ABB RobotStudio station: Modulo_1.rspag

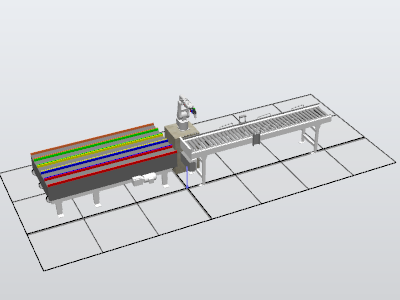
--- station ---
Station Prototipo1 (saved by RobotStudio 25.1.11133.0)
Controller Controlador1, task T_ROB1: task frame (RAPID world) sits at (289.3, 766.92, 800) mm, rotated rx 0 ry 0 rz -90 deg in the station
Controller Controlador1
  mechanical unit ROB_1: Robot1, 6 joints, base frame (0, 0, 0) mm
Layout (positions relative to the parent item):
  - Cinta entrada [part, from %ABB.RobotStudio.Models.Conveyors%\Conveyor Guide 400.rslib] at (77.15, 0, 0) mm
  - Apoyo1 [part], size 500 x 500 x 800 mm
  - Robot1 [mechanism, from %ABB.RobotStudio.Models.IRB120%\IRB120_3_58_G_01.rslib] at (289.3, 766.92, 800) mm, rotated rx 0 ry 0 rz -90 deg; joint values [0, 0, 0, 0, 0.5236, 0] (rad or m)
  - Apoyo cinta salida [part, from %ABB.RobotStudio.Models.Conveyors%\Conveyor 2400 3str h2.rslib] at (-191.15, 1159.17, 0) mm, rotated rx 0 ry 0 rz 180 deg
  - Estropajo_base [part] at (2748.27, 147.09, 782.53) mm, size 80 x 120 x 43 mm
  - Source [smart component, from Components\Source.rslib]
      properties: Source=Estropajo_base; Copy=(none); Parent=(none); Position=[2.748273 0.147093 0.782531]; Orientation=[0 0 0]; Transient=true; PhysicsBehavior=-1
  - LinearMover2 [smart component, from Components\LinearMover2.rslib]
      properties: Object=(none); Direction=[-1 0 0]; Distance=2.5; Duration=3; Reference=Global; ReferenceObject=(none)
  - Sink [smart component, from Components\Sink.rslib]
      properties: Object=(none)
  - Source_2 [smart component, from Components\Source.rslib]
      properties: Source=Estropajo_azul; Copy=(none); Parent=(none); Position=[2.748273 0.147093 0.782531]; Orientation=[0 0 0]; Transient=true; PhysicsBehavior=-1
  - Estropajo_azul [part] at (2748.27, 147.09, 782.53) mm, size 80 x 120 x 43 mm
  - Source_3 [smart component, from Components\Source.rslib]
      properties: Source=Estropajo_naranja; Copy=(none); Parent=(none); Position=[2.748273 0.147093 0.782531]; Orientation=[0 0 0]; Transient=true; PhysicsBehavior=-1
  - Source_4 [smart component, from Components\Source.rslib]
      properties: Source=Estropajo_amarillo; Copy=(none); Parent=(none); Position=[2.748273 0.147093 0.782531]; Orientation=[0 0 0]; Transient=true; PhysicsBehavior=-1
  - Source_6 [smart component, from Components\Source.rslib]
      properties: Source=Estropajo_verde; Copy=(none); Parent=(none); Position=[2.748273 0.147093 0.782531]; Orientation=[0 0 0]; Transient=true; PhysicsBehavior=-1
  - Estropajo_amarillo [part] at (2748.27, 147.09, 782.53) mm, size 80 x 120 x 43 mm
  - Estropajo_naranja [part] at (2748.27, 147.09, 782.53) mm, size 80 x 120 x 43 mm
  - Estropajo_verde [part] at (2748.27, 147.09, 782.53) mm, size 80 x 120 x 43 mm
  - Estropajo_5 [part] at (248.27, 147.09, 782.53) mm, size 80 x 120 x 43 mm
  - Estropajo_6 [part] at (-216.02, 245.91, 691.61) mm, size 80 x 120 x 43 mm
  - MyTool [mechanism, from Training Objects\myTool.rslib] at (289.3, 402.56, 1394) mm, rotated rx 180 ry 60 rz 90 deg
  - Attacher [smart component, from Components\Attacher.rslib]
      properties: Parent=MyTool; Flange=0; Child=(none); Mount=false; Offset=[0 0 0]; Orientation=[0 0 0]
  - Detacher [smart component, from Components\Detacher.rslib]
      properties: Child=(none); KeepPosition=true
  - Attacher_2 [smart component, from Components\Attacher.rslib]
      properties: Parent=MyTool; Flange=0; Child=(none); Mount=false; Offset=[0 0 0]; Orientation=[0 0 0]
  - Attacher_3 [smart component, from Components\Attacher.rslib]
      properties: Parent=MyTool; Flange=0; Child=(none); Mount=false; Offset=[0 0 0]; Orientation=[0 0 0]
  - Attacher_4 [smart component, from Components\Attacher.rslib]
      properties: Parent=MyTool; Flange=0; Child=(none); Mount=false; Offset=[0 0 0]; Orientation=[0 0 0]
  - Attacher_5 [smart component, from Components\Attacher.rslib]
      properties: Parent=MyTool; Flange=0; Child=(none); Mount=false; Offset=[0 0 0]; Orientation=[0 0 0]
  - LinearMover2_2 [smart component, from Components\LinearMover2.rslib]
      properties: Object=(none); Direction=[-1 0 0]; Distance=2.2; Duration=3; Reference=Global; ReferenceObject=(none)
  - Cinta entrada [part, from Components\Cinta salida.rslib] at (100, -50, 0) mm
Attachment: MyTool is attached to Robot1 / Link6
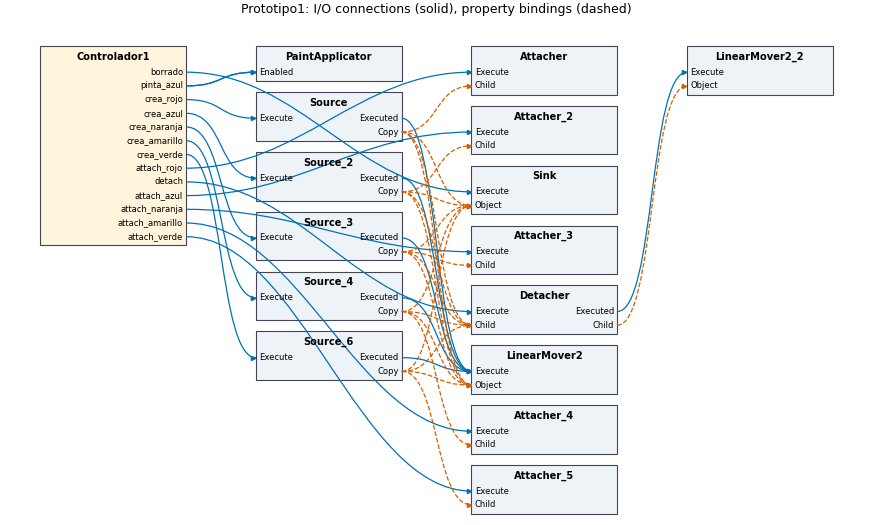
Station logic (signal -> signal, property => property):
  Source.Executed -> LinearMover2.Execute
  Controlador1.borrado -> Sink.Execute
  Controlador1.pinta_azul -> PaintApplicator.Enabled
  Controlador1.pinta_azul -> PaintApplicator_2.Enabled
  Source_2.Executed -> LinearMover2.Execute
  Source_3.Executed -> LinearMover2.Execute
  Source_4.Executed -> LinearMover2.Execute
  Controlador1.crea_rojo -> Source.Execute
  Controlador1.crea_azul -> Source_2.Execute
  Controlador1.crea_naranja -> Source_3.Execute
  Controlador1.crea_amarillo -> Source_4.Execute
  Controlador1.crea_verde -> Source_6.Execute
  Source_6.Executed -> LinearMover2.Execute
  Controlador1.attach_rojo -> Attacher.Execute
  Controlador1.detach -> Detacher.Execute
  Controlador1.attach_azul -> Attacher_2.Execute
  Controlador1.attach_naranja -> Attacher_3.Execute
  Controlador1.attach_amarillo -> Attacher_4.Execute
  Controlador1.attach_verde -> Attacher_5.Execute
  Detacher.Executed -> LinearMover2_2.Execute
  Source.Copy => Sink.Object
  Source.Copy => LinearMover2.Object
  Source_2.Copy => LinearMover2.Object
  Source_2.Copy => Sink.Object
  Source_3.Copy => Sink.Object
  Source_4.Copy => Sink.Object
  Source_3.Copy => LinearMover2.Object
  Source_4.Copy => LinearMover2.Object
  Source_6.Copy => LinearMover2.Object
  Source_6.Copy => Sink.Object
  Source.Copy => Attacher.Child
  Source.Copy => Detacher.Child
  Source_2.Copy => Detacher.Child
  Source_4.Copy => Detacher.Child
  Source_6.Copy => Detacher.Child
  Source_3.Copy => Detacher.Child
  Source_2.Copy => Attacher_2.Child
  Source_3.Copy => Attacher_3.Child
  Source_4.Copy => Attacher_4.Child
  Source_6.Copy => Attacher_5.Child
  Detacher.Child => LinearMover2_2.Object

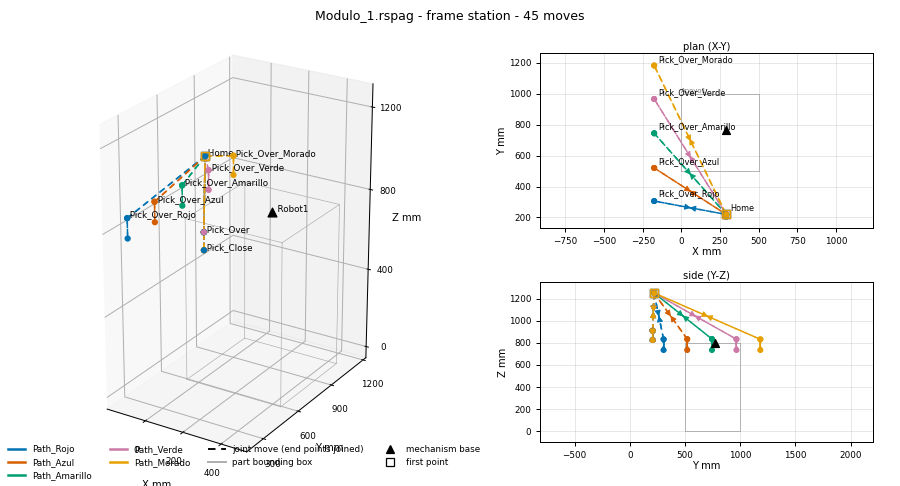
[picture p0: tool path of Modulo_1.rspag in frame station, 45 of 45 moves have a stored position in this frame; points joined in program order, loops and branches not executed]
--- Controller Data/Controlador1/RAPID/TASK1/PROGMOD/CalibData.mod ---
MODULE CalibData
    PERS tooldata MyTool:=[TRUE,[[31.792631019,0,229.638935148],[0.945518576,0,0.325568154,0]],[1,[0,0,1],[1,0,0,0],0,0,0]];
ENDMODULE

--- Controller Data/Controlador1/RAPID/TASK1/PROGMOD/Module1.mod ---
MODULE Module1
    CONST robtarget Home:=[[547.330665099,0,451.64730631],[0.190808996,0,0.981627183,0],[-1,0,-1,0],[9E+09,9E+09,9E+09,9E+09,9E+09,9E+09]];
    CONST robtarget Pick_Over:=[[559.825628438,-1.031837605,109.196112849],[0,0,1,0],[-1,0,-1,0],[9E+09,9E+09,9E+09,9E+09,9E+09,9E+09]];
    CONST robtarget Pick_Close:=[[559.825628438,-1.031837605,25.531],[0,0,1,0],[-1,-1,0,1],[9E+09,9E+09,9E+09,9E+09,9E+09,9E+09]];
    CONST robtarget Pick_Over_Rojo:=[[461.009628438,-465.329837605,32.056284824],[0,0.707106781,0.707106781,0],[-1,-1,0,0],[9E+09,9E+09,9E+09,9E+09,9E+09,9E+09]];
    CONST robtarget Pick_Close_Rojo:=[[461.009628438,-465.329837605,-65.385],[0,0.707106781,0.707106781,0],[-1,-1,1,0],[9E+09,9E+09,9E+09,9E+09,9E+09,9E+09]];
    CONST robtarget Pick_Over_Azul:=[[246.918628438,-465.329837605,33.65920877],[0,0.707106781,0.707106781,0],[-1,-1,1,0],[9E+09,9E+09,9E+09,9E+09,9E+09,9E+09]];
    CONST robtarget Pick_Close_Azul:=[[246.918628438,-465.329837605,-65.385],[0,0.707106781,0.707106781,0],[-1,-2,1,0],[9E+09,9E+09,9E+09,9E+09,9E+09,9E+09]];
    CONST robtarget Pick_Over_Amarillo:=[[23.13670375,-465.329837605,34.646672212],[0,0.707106781,0.707106781,0],[-1,0,-1,1],[9E+09,9E+09,9E+09,9E+09,9E+09,9E+09]];
    CONST robtarget Pick_Close_Amarillo:=[[23.13670375,-465.329837605,-65.385],[0,0.707106781,0.707106781,0],[-1,0,-1,1],[9E+09,9E+09,9E+09,9E+09,9E+09,9E+09]];
    CONST robtarget Pick_Over_Verde:=[[-198.51110118,-465.329837605,33.114552001],[0,0.707106781,0.707106781,0],[-2,1,-2,0],[9E+09,9E+09,9E+09,9E+09,9E+09,9E+09]];
    CONST robtarget Pick_Close_Verde:=[[-198.51110118,-465.329837605,-65.385],[0,0.707106781,0.707106781,0],[-2,1,-2,0],[9E+09,9E+09,9E+09,9E+09,9E+09,9E+09]];
    CONST robtarget Pick_Over_Morado:=[[-414.848394347,-465.329837605,31.927230483],[0,0.707106781,0.707106781,0],[-2,0,-2,0],[9E+09,9E+09,9E+09,9E+09,9E+09,9E+09]];
    CONST robtarget Pick_Close_Morado:=[[-414.848394347,-465.329837605,-65.385],[0,0.707106781,0.707106781,0],[-2,0,-2,0],[9E+09,9E+09,9E+09,9E+09,9E+09,9E+09]];
    VAR socketdev ServerSocket;
    VAR socketdev ClientSocket;
    VAR socketdev ServerSocket_fin_mov;
    VAR socketdev ClientSocket_fin_mov;
    VAR socketdev ServerSocket_fin_total;
    VAR socketdev ClientSocket_fin_total;
    VAR bool ejecutar := TRUE;
    VAR string senyalStr;
    VAR num senyalNum;
    VAR bool Ok;
    VAR num Valor;

    PROC main()
        !Add your code here
        VAR num myrandom;
        VAR num n;
        SocketCreate serverSocket;
        SocketBind serverSocket, "127.0.0.1", 8000;
        SocketListen serverSocket;
        SocketAccept serverSocket, clientSocket, \Time:=WAIT_MAX;
        SocketSend clientSocket \str:="Conexion con abb correcta.";


        WaitTime 5;
        !Ok:= StrToVal(senyalStr,senyalNum);
        FOR n FROM 1 TO 5 DO
            myrandom := (Rand() MOD 5) + 1;


            IF myrandom=1 THEN
                PulseDO crea_rojo;
                 WaitTime 3;
            ELSEIF myrandom=2 THEN
                PulseDO crea_azul;
                WaitTime 3;
            ELSEIF myrandom=3 THEN
                PulseDO crea_naranja;
                WaitTime 3;
            ELSEIF myrandom=4 THEN
                PulseDO crea_amarillo;
                WaitTime 3;
            ELSEIF myrandom=5 THEN
                PulseDO crea_verde;
                WaitTime 3;
            ENDIF

            !hacer aqui que mande una señal al python para que empiece a ver el color
            SocketSend clientSocket \str:="Activa vision";

            SocketReceive ClientSocket \str:=senyalStr;
            IF senyalStr = "Rojo" THEN
                Path_Rojo;
                WaitTime 3;
                PulseDO borrado;
            ELSEIF senyalStr = "Verde" THEN
                Path_Verde;
                WaitTime 3;
                PulseDO borrado;
            ELSEIF senyalStr = "Azul" THEN
                Path_Azul;
                WaitTime 3;
                PulseDO borrado;
            ELSEIF senyalStr = "Amarillo" THEN
                Path_Amarillo;
                WaitTime 3;
                PulseDO borrado;
            ELSEIF senyalStr = "Naranja" THEN
                Path_Morado;
                WaitTime 3;
                PulseDO borrado;

           ENDIF





        ENDFOR
        PulseDO borrado;
    ENDPROC
    PROC Path_Rojo()
        MoveJ Home,v1000,fine,MyTool\WObj:=wobj0;
        MoveJ Pick_Over,v1000,fine,MyTool\WObj:=wobj0;
        MoveJ Pick_Close,v300,fine,MyTool\WObj:=wobj0;
        PulseDO attach_rojo;
        MoveJ Pick_Over,v300,fine,MyTool\WObj:=wobj0;

        MoveJ Home,v1000,fine,MyTool\WObj:=wobj0;
        MoveJ Pick_Over_Rojo,v1000,fine,MyTool\WObj:=wobj0;
        MoveJ Pick_Close_Rojo,v300,fine,MyTool\WObj:=wobj0;
        PulseDO detach;
        MoveJ Pick_Over_Rojo,v1000,fine,MyTool\WObj:=wobj0;
        MoveJ Home,v1000,fine,MyTool\WObj:=wobj0;
    ENDPROC
    PROC Path_Azul()
        MoveJ Home,v1000,fine,MyTool\WObj:=wobj0;
        MoveJ Pick_Over,v1000,fine,MyTool\WObj:=wobj0;
        MoveJ Pick_Close,v300,fine,MyTool\WObj:=wobj0;
        PulseDO attach_azul;
        MoveJ Pick_Over,v1000,fine,MyTool\WObj:=wobj0;

        MoveJ Home,v1000,fine,MyTool\WObj:=wobj0;
        MoveJ Pick_Over_Azul,v1000,fine,MyTool\WObj:=wobj0;
        MoveJ Pick_Close_Azul,v300,fine,MyTool\WObj:=wobj0;
        PulseDO detach;
        MoveJ Pick_Over_Azul,v1000,fine,MyTool\WObj:=wobj0;
        MoveJ Home,v1000,fine,MyTool\WObj:=wobj0;
    ENDPROC
    PROC Path_Amarillo()
        MoveJ Home,v1000,fine,MyTool\WObj:=wobj0;
        MoveJ Pick_Over,v1000,fine,MyTool\WObj:=wobj0;
        MoveJ Pick_Close,v300,fine,MyTool\WObj:=wobj0;
        PulseDO attach_amarillo;
        MoveJ Pick_Over,v1000,fine,MyTool\WObj:=wobj0;

        MoveJ Home,v1000,fine,MyTool\WObj:=wobj0;
        MoveJ Pick_Over_Amarillo,v1000,fine,MyTool\WObj:=wobj0;
        MoveJ Pick_Close_Amarillo,v300,fine,MyTool\WObj:=wobj0;
        PulseDO detach;
        MoveJ Pick_Over_Amarillo,v1000,fine,MyTool\WObj:=wobj0;
        MoveJ Home,v1000,fine,MyTool\WObj:=wobj0;
    ENDPROC
    PROC Path_Verde()
        MoveJ Home,v1000,fine,MyTool\WObj:=wobj0;
        MoveJ Pick_Over,v1000,fine,MyTool\WObj:=wobj0;
        MoveJ Pick_Close,v300,fine,MyTool\WObj:=wobj0;
        PulseDO attach_verde;
        MoveJ Pick_Over,v1000,fine,MyTool\WObj:=wobj0;

        MoveJ Home,v1000,fine,MyTool\WObj:=wobj0;
        MoveJ Pick_Over_Verde,v1000,fine,MyTool\WObj:=wobj0;
        MoveJ Pick_Close_Verde,v300,fine,MyTool\WObj:=wobj0;
        PulseDO detach;
        MoveJ Pick_Over_Verde,v1000,fine,MyTool\WObj:=wobj0;
        MoveJ Home,v1000,fine,MyTool\WObj:=wobj0;
    ENDPROC
    PROC Path_Morado()
        MoveJ Home,v1000,fine,MyTool\WObj:=wobj0;
        MoveJ Pick_Over,v1000,fine,MyTool\WObj:=wobj0;
        MoveJ Pick_Close,v300,fine,MyTool\WObj:=wobj0;
        PulseDO attach_naranja;
        MoveJ Pick_Over,v1000,fine,MyTool\WObj:=wobj0;

        MoveJ Home,v1000,fine,MyTool\WObj:=wobj0;
        MoveJ Pick_Over_Morado,v1000,fine,MyTool\WObj:=wobj0;
        MoveJ Pick_Close_Morado,v300,fine,MyTool\WObj:=wobj0;
        PulseDO detach;
        MoveJ Pick_Over_Morado,v1000,fine,MyTool\WObj:=wobj0;
        MoveJ Home,v1000,fine,MyTool\WObj:=wobj0;
    ENDPROC
ENDMODULE

--- Controller Data/Controlador1/SYSPAR/EIO.cfg ---
EIO:CFG_1.0:6:1::
#
EIO_SIGNAL:

      -Name "crea_rojo" -SignalType "DO" -Access "All"

      -Name "crea_azul" -SignalType "DO" -Access "All"

      -Name "crea_verde" -SignalType "DO" -Access "All"

      -Name "crea_amarillo" -SignalType "DO" -Access "All"

      -Name "crea_naranja" -SignalType "DO" -Access "All"

      -Name "borrado" -SignalType "DO" -Access "All"

      -Name "attach_rojo" -SignalType "DO" -Access "All"

      -Name "attach_verde" -SignalType "DO" -Access "All"

      -Name "attach_amarillo" -SignalType "DO" -Access "All"

      -Name "attach_azul" -SignalType "DO" -Access "All"

      -Name "attach_naranja" -SignalType "DO" -Access "All"

      -Name "detach" -SignalType "DO" -Access "All"
